// Mitsubishi GX Works2 project: LRI - inclusão de RESET (RST)   PLC: Q03UDV
// HelloWorld

PROGRAM MAIN
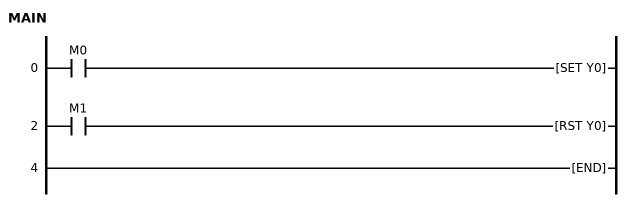
0     LD      M0
      SET     Y0
2     LD      M1
      RST     Y0
4     END
END_PROGRAM
